% RSLogix 500 project Ladder logic code file.RSS, saved by version 8.30.00.15 %
PROJECT "UNTITLED"    % processor: SLC 500, 1747-L531 %

PROGRAM FILES
  LAD 2 "MAIN"  4 rungs
  LAD 3 "SAFETY"  3 rungs
  LAD 5 "GAS + IGIN"  4 rungs  % Routine for gas value and ignitier %
  LAD 6 "ERROR"  6 rungs  % Flame not igniting error %

DATA FILES
  O0 OUTPUT  2 elements
  I1 INPUT  2 elements
  S2 STATUS  83 elements
  B3 BINARY  2 elements
  T4 TIMER  3 elements
  C5 COUNTER  1 elements
  R6 CONTROL  1 elements
  N7 INTEGER  11 elements
  F8 FLOAT  1 elements

LADDER 2 "MAIN"
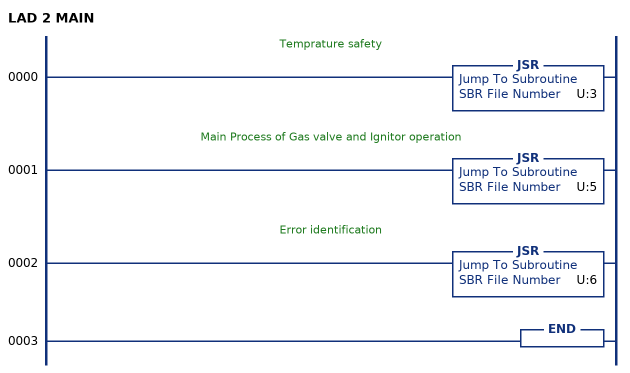
% Rung: 0 %  % edit flag set %
% Temprature safety %
SOR JSR U:3 EOR
% Rung: 1 %
% Main Process of Gas valve and Ignitor operation %
SOR JSR U:5 EOR
% Rung: 2 %
% Error identification %
SOR JSR U:6 EOR
% Rung: 3 %
SOR END EOR

LADDER 3 "SAFETY"
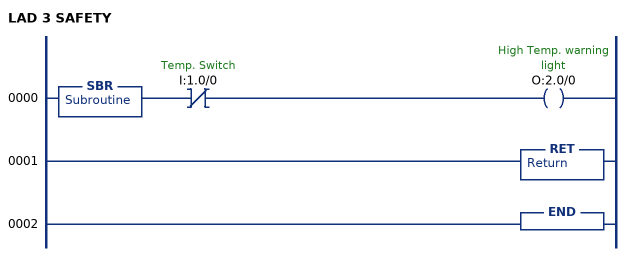
% Rung: 0 %  % edit flag set %
SOR SBR XIO I:1.0/0 OTE O:2.0/0 EOR
%   I:1.0/0  "Temp. Switch" %
%   O:2.0/0  "High Temp. warning light" %
% Rung: 1 %
SOR RET EOR
% Rung: 2 %
SOR END EOR

LADDER 5 "GAS + IGIN"    % Routine for gas value and ignitier %
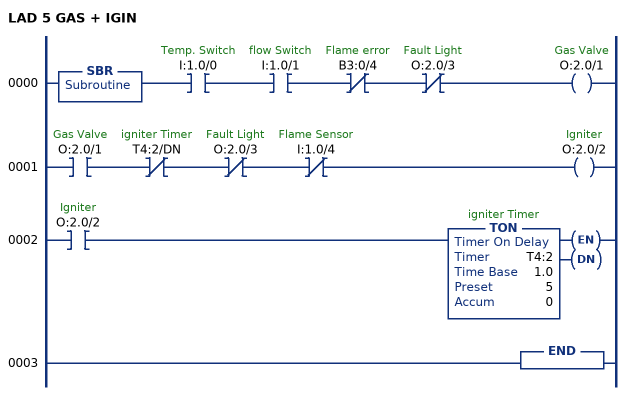
% Rung: 0 %
SOR SBR XIC I:1.0/0 XIC I:1.0/1 XIO B3:0/4 XIO O:2.0/3 OTE O:2.0/1 EOR
%   I:1.0/0  "Temp. Switch" %
%   I:1.0/1  "flow Switch" %
%   B3:0/4  "Flame error" %
%   O:2.0/3  "Fault Light" %
%   O:2.0/1  "Gas Valve" %
% Rung: 1 %
SOR XIC O:2.0/1 XIO T4:2/DN XIO O:2.0/3 XIO I:1.0/4 OTE O:2.0/2 EOR
%   O:2.0/1  "Gas Valve" %
%   T4:2  "igniter Timer" %
%   O:2.0/3  "Fault Light" %
%   I:1.0/4  "Flame Sensor" %
%   O:2.0/2  "Igniter" %
% Rung: 2 %
SOR XIC O:2.0/2 TON T4:2 1.0 5 0 EOR
%   O:2.0/2  "Igniter" %
%   T4:2  "igniter Timer" %
% Rung: 3 %
SOR END EOR

LADDER 6 "ERROR"    % Flame not igniting error %
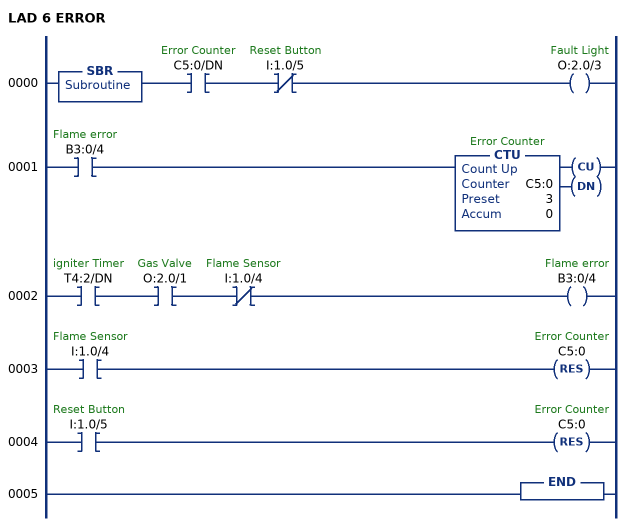
% Rung: 0 %
SOR SBR XIC C5:0/DN XIO I:1.0/5 OTE O:2.0/3 EOR
%   C5:0  "Error Counter" %
%   I:1.0/5  "Reset Button" %
%   O:2.0/3  "Fault Light" %
% Rung: 1 %
SOR XIC B3:0/4 CTU C5:0 3 0 EOR
%   B3:0/4  "Flame error" %
%   C5:0  "Error Counter" %
% Rung: 2 %
SOR XIC T4:2/DN XIC O:2.0/1 XIO I:1.0/4 OTE B3:0/4 EOR
%   T4:2  "igniter Timer" %
%   O:2.0/1  "Gas Valve" %
%   I:1.0/4  "Flame Sensor" %
%   B3:0/4  "Flame error" %
% Rung: 3 %
SOR XIC I:1.0/4 RES C5:0 EOR
%   I:1.0/4  "Flame Sensor" %
%   C5:0  "Error Counter" %
% Rung: 4 %
SOR XIC I:1.0/5 RES C5:0 EOR
%   I:1.0/5  "Reset Button" %
%   C5:0  "Error Counter" %
% Rung: 5 %
SOR END EOR

OTHER DOCUMENTED ADDRESSES
  T4:0/DN  T4

DATA TABLE (non-zero values as saved)
DATA B3
% B3:0 % 0X0001 0X0000
DATA T4
% .PRE .ACC %
% T4:0 % 20 20
% T4:2 % 5 0
DATA C5
% .PRE .ACC %
% C5:0 % 3 0
